{attribute 'pack_mode' := '2'}
TYPE ST_INSTANCE_CTRL :
STRUCT
  Cmd     : E_INSTANCE_CMD;
END_STRUCT
END_TYPE

(* stored: Version 1.1.0.1
   DUT ST_INSTANCE_CTRL: Id {cec64f75-8d37-4a85-9e3c-06086ef2adb2} *)
